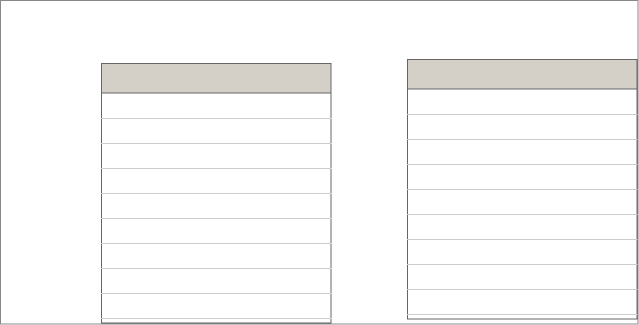
VISUALIZATION EM  // 639x325
    Table (101,63 230x260), data array: Unit01.EM_Resetting_Done
        p3854506369: Unit01.EM_Resetting_Done[INDEX]
    Table (407,59 230x260), data array: Unit02.EM_Resetting_Done
        p3854506369: Unit02.EM_Resetting_Done[INDEX]
END_VISUALIZATION

(* stored: Version 1.1.0.1, ProductVersion 3.1.4022.16
   Visu EM: Id {6ccb4c15-9ce0-4de7-b183-c485c7a31d36} *)
